PROGRAM PRG_CASE_FinaliseDataManual
VAR
	fbCase_FinaliseData		: FB_CASE_FinaliseData;
	
	(* Init function/method declarations*)
	rTrigDataInit		: R_TRIG;
	bDataInit			: BOOL;
	iOuter				: INT;
	iPack				: INT;
	sPackNum			: STRING;
	sOuterNum			: STRING;
	sPackCode			: STRING;
	
	(* Inputs *)
	bExecute 				: BOOL;		(* set TRUE to move Outers *)
	bDoorReject				: BOOL;
	stRejectReasonsForCase	: ST_RejectReasonsForCase;
	
	(* In/Out *)
	stProductInstruction	: ST_PCM_Status;
	stCodeInfo_Outer		: ST_CodeInfo;
	stCACData 				: ST_CAC_Data;	(* Case Queue *)
	stCACDataHMI			: ST_HMI_CAC_Data;
	
	(* Outputs *)
	bDone 					: BOOL;
	bBusy					: BOOL;

	bCACValid				: BOOL;
	bCACInvalid				: BOOL;

	bCheckDuplicates		: BOOL;
	bReadyToValidate		: BOOL;
	
	sRejectCode				: T_MaxString;
	sCaseContent			: T_LongSTRING;
	
END_VAR

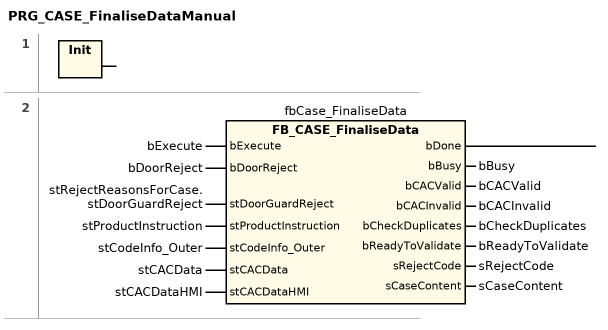
// NETWORK 1
Init();

// NETWORK 2
fbCase_FinaliseData(
    bExecute := bExecute,
    bDoorReject := bDoorReject,
    stDoorGuardReject := stRejectReasonsForCase.stDoorGuardReject,
    stProductInstruction := stProductInstruction,
    stCodeInfo_Outer := stCodeInfo_Outer,
    stCACData := stCACData,
    stCACDataHMI := stCACDataHMI,
    bBusy => bBusy,
    bCACValid => bCACValid,
    bCACInvalid => bCACInvalid,
    bCheckDuplicates => bCheckDuplicates,
    bReadyToValidate => bReadyToValidate,
    sRejectCode => sRejectCode,
    sCaseContent => sCaseContent); // FB_CASE_FinaliseData

ACTION Init:

rTrigDataInit(CLK := bDataInit);

IF rTrigDataInit.Q THEN
	
stProductInstruction.nOutersPerCase		:= 50;
stProductInstruction.nPacksPerOuter 	:= 10;

	FOR iOuter := 1 TO stProductInstruction.nOutersPerCase DO
		(* Outer number z zerami *)
		sOuterNum := F_StringAddPrefix(INT_TO_STRING(iOuter),2,'0');
		
		(* Write Outers barcodes *)
		stCACData.Outer[iOuter].Barcode    := CONCAT('OUTER', sOuterNum);
		stCACData.Outer[iOuter].OuterCodeStatus := 5;
		stCACData.Outer[iOuter].OuterRejectCode := 'OK';
		
		FOR iPack := 1 TO stProductInstruction.nPacksPerOuter DO
			(* Pack number dwucyfrowy z zerami *)
			sPackNum := F_StringAddPrefix(INT_TO_STRING(iPack),2,'0');			
			(* Sklej pack code *)
			sPackCode := CONCAT(CONCAT('PACK', sPackNum), CONCAT('OUTER', sOuterNum));
			
			(* Write Pack Barcodes / Data*)
			stCACData.Outer[iOuter].PackCode[iPack]			:= sPackCode;
			stCACData.Outer[iOuter].PackCodeStatus[iPack]	:= 5;
			stCACData.Outer[iOuter].PackRejectID[iPack]		:= 0;			
			stCACData.Outer[iOuter].PackRejectCode[iPack]	:= 'OK';
			
						
			stCACData.Outer[iOuter].NumberOfPacks := stProductInstruction.nPacksPerOuter;
			
		END_FOR;
	END_FOR;	

//initialize needed data structures
stCACData.NumberOfOuters						:= stProductInstruction.nOutersPerCase;
stCACData.CaseRejectCode						:= 'OK';
stCodeInfo_Outer.nEntireLength					:= 7;
stCodeInfo_Outer.stSerialCode.nCodeStartPos 	:= 1;
stCodeInfo_Outer.stSerialCode.nCodeLength 		:= 7;
stCACData.Barcode 								:= 'CaseBarcode';
	
END_IF
END_ACTION

END_PROGRAM

(* stored: Version 1.1.0.1
   POU PRG_CASE_FinaliseDataManual: Id {de1c4946-2f6a-46af-94e8-69091e414096}, SpecialFunc None
   Action Init: Id {08194a4d-05fa-4272-8ec8-ee3a74e4e1b9} *)
